TYPE EL2008 :
STRUCT
	// 8ch. Digital Output Slot
	e2008	AT %Q*	: BYTE;
END_STRUCT
END_TYPE

(* stored: Version 1.1.0.1, ProductVersion 3.1.4024.12
   DUT EL2008: Id {da58d72c-0bc7-4574-9e96-e87a45fbbf41} *)
